FUNCTION_BLOCK FB_EpicsInOutPMPS EXTENDS FB_EpicsInOut
VAR_IN_OUT
    fbArbiter: FB_Arbiter;
    fbFFHWO: FB_HardwareFFOutput;
END_VAR
VAR_INPUT
    stTransitionBeam: ST_BeamParams := PMPS_GVL.cstSafeBeam;
    nTransitionAssertionID: UDINT;
END_VAR
VAR
    fbStatePMPS: FB_PositionStatePMPS;
    fbEncErrFFO: FB_EncErrorFFO;
END_VAR

SUPER^(stMotionStage:=stMotionStage,
       stOut:=stOut,
       stIn:=stIn,
       bEnable:=bEnable,
       enumSet:=enumSet,
       bError=>bError,
       nErrorId=>nErrorId,
       sErrorMessage=>sErrorMessage,
       bBusy=>bBusy,
       bDone=>bDone,
       enumGet=>enumGet);

fbStatePMPS(fbArbiter:=fbArbiter,
            fbFFHWO:=fbFFHWO,
            stMotionStage:=stMotionStage,
            arrStates:=arrStates,
            bRequestTransition:=bBusy,
            setState:=enumSet,
            getState:=enumGet,
            nTransitionAssertionID:=nTransitionAssertionID);

fbEncErrFFO(
    stMotionStage:=stMotionStage,
    fbFFHWO:=fbFFHWO,
    bAutoReset:=TRUE);

END_FUNCTION_BLOCK

(* stored: Version 1.1.0.1, ProductVersion 3.1.4022.18
   POU FB_EpicsInOutPMPS: Id {aa945542-c9b2-4cf9-a365-9f97c65083b0}, SpecialFunc None *)
